INTERFACE I_HE_SATT_FindOptimalFilterCombination


METHOD PUBLIC FindOptimalCombination
VAR_INPUT
    fPhotonEnergy_eV : LREAL;
	(* [0.0 - 1.0]*)
	fRequestedTransmission	: LREAL;
	eRequestedRoundingMode	: E_HE_SATT_RoundingMode;
	fRequestedAllowableTolerance	: LREAL;
    iFilterCombinationCollector : I_HE_SATT_FilterCombinationCollector;
END_VAR
VAR_OUTPUT
    iOptimalFilterCombination : I_HE_SATT_FilterCombination;
END_VAR
END_METHOD


PROPERTY Status : REFERENCE TO ST_HE_SATT_Status
GET
END_GET
END_PROPERTY

END_INTERFACE

(* stored: Version 1.1.0.1
   Itf I_HE_SATT_FindOptimalFilterCombination: Id {71a4134d-dc69-4439-95ed-acfd41c0007d}
   Method FindOptimalCombination: Id {88e23ce1-0e8c-4bc9-8b84-c2597bd7af2f}
   Property Status: Id {200598b7-4f17-4e4c-ace5-5ba4a0cb7ab0}
   Get Get: Id {0c7cc512-3f9c-4c5f-9a29-18fb192bcc89} *)
